TYPE E_InstrumentUsage :
(
	InstruUsage_UNKNOWM := 0,
	InstruUsage_ClinicalUsed := 1,
	InstruUsage_TestUsed := 2,
	InstruUsage_InstruSell := 3,
	InstruUsage_Training := 4
);
END_TYPE

(* stored: Version 1.1.0.1, ProductVersion 3.1.4024.11
   DUT E_InstrumentUsage: Id {d2832e37-0a58-42c1-a092-df9e94583ca0} *)
